(* Logix 5000 project; controller TrayLoader_EnSG vendor 1 type 14 code 156 rev 32.11; software revision 32.02; part 2 of 3 *)
(* tags used below, declared in another part *)
   blink1s : BOOL;
   Emergency : BOOL;
   Feeder_st : INT;
   FeedMotionCtrl : MOTION_INSTRUCTION;
   modRes : INT;
   mot_conv_in : INT;   // Conveyor Motor
   oddEven : BOOL;
   ons : DINT;
   ons5 : INT;
   srvMASRTray : BOOL;
   SrvMoveType : DINT;
   TrayAxis_pos : DINT;   // servo position increment
   TrayMotionCtrl : MOTION_INSTRUCTION;
   UpLift_forward : BOOL;
   UpLift_start : BOOL;
   UpLift_stop : BOOL;
   Auto : BOOL;
   auto_resumeFeeder : BOOL;
   corr_elapsedTrayPos : DINT;
   DecelDelay_t : TIMER;
   DecelVal : DINT;
   delta_TrayActualPos : DINT;
   dummy1 : BOOL;
   elapsedTrayPos : DINT;
   enableCheckingMsg : MESSAGE;
   enableHwOvertravelMsg : MESSAGE;
   EnableInputChecking : DINT;
   Fault : BOOL;
   feed_decel_spd : INT;   // mcd speed
   Feed_st : INT;
   feedDela_t : TIMER;
   FeederConvAxis : AXIS_CIP_DRIVE;
   FeedSpeed : DINT;
   finishPush_t : TIMER;
   finishPush_t0 : TIMER;
   hmi_Reset : BOOL;
   hmi_resetTrayCtr : BOOL;
   hmi_setSpeedRef : DINT;
   hmi_setSpeedRef100 : INT;
   JogPulse_m : BOOL;
   JogTime : TIMER;
   lastActualPosUnit : DINT;
   lineCtr : INT;
   man_disableUplift : BOOL;
   man_engageClutch : BOOL;
   man_feederReload : BOOL;
   man_FeedRailEnd : BOOL;
   man_JogLineDown : BOOL;
   man_JogLineUp : BOOL;
   man_ledRun : BOOL;
   man_ledStart : BOOL;
   man_ledWarning : BOOL;
   man_mot_conv_in0 : BOOL;
   man_mot_conv_in1 : BOOL;
   man_mot_conv_in2 : BOOL;
   man_mot_conv_in3 : BOOL;
   man_mot_conv_in4 : BOOL;
   man_mot_upLiftBrake : BOOL;
   man_sol_engageClutch : BOOL;
   man_SrvTrayJogMotorFwd : BOOL;
   man_srvTrayStop : BOOL;
   man_sv_exit : BOOL;
   man_sv_flipperIn : BOOL;
   man_sv_flipperOut : BOOL;
   man_sv_gripper : BOOL;
   man_sv_gripperArm : BOOL;
   man_sv_tray_in : BOOL;
   man_sv_tray_out : BOOL;
   man_UpLift_forward : BOOL;
   man_UpLift_start : BOOL;
   mot_upLiftBrake : BOOL;
   nc_ls_UpLift_bot : BOOL;
   nc_ls_UpLift_top : BOOL;
   nc_ps_exit : BOOL;   // indicate Full exit qeue
   negStepPulse : DINT;
   no_ps_FeedPlankHome : BOOL;
   no_ps_FeedRailDecel : BOOL;
   no_ps_FeedRailEndEven : BOOL;   // ps on end of FeederRail
   no_ps_FeedRailEndOdd : BOOL;
   no_ps_Serp_top : BOOL;   // ps serpentine top
   ons4 : INT;
   ons6 : DINT;
   ons7 : DINT;
   pauseFeeder : BOOL;
   ps_serp_top_t : TIMER;
   ps_serp_top_tof : TIMER;
   RailDecel : BOOL;
   Recover_UpLift : BOOL;
   ref_elpasedTrayPos : DINT;
   Reset : BOOL;
   resumeFeeder : BOOL;
   rs_sv_exit_top : BOOL;
   rs_sv_flipperOut_top : BOOL;
   rs_sv_tray_out_bot : BOOL;
   Run : BOOL;
   RunOff_t : TIMER;
   RunOn_t : TIMER;
   serp_top_t_pre : DINT;
   serp_top_tof_pre : DINT;
   ServoEndRun : BOOL;
   ServoEndRunPulse : BOOL;
   sol_engageClutch : BOOL;
   SrvTrayJogMot : BOOL;
   SrvTrayStep : BOOL;   // Servo Tray Step down
   SrvTrayStop : BOOL;
   StartSpeed : DINT;
   stepPulse : DINT;
   stepPulseAct : DINT;
   sv_exit : BOOL;
   sv_flipperIn : BOOL;
   sv_flipperOut : BOOL;
   sv_flipperOut_bot : BOOL;
   sv_flipperOut_top : BOOL;
   sv_gripper : BOOL;
   sv_gripper_bot : BOOL;   // pneu gripper
   sv_gripper_top : BOOL;
   sv_gripperArm : BOOL;
   sv_tray_in : BOOL;
   sv_tray_out : BOOL;
   sysStop : BOOL;
   total_tray : DINT;
   TrayAxis : AXIS_CIP_DRIVE;
   TraySrvBreakU : BOOL;
   TrayWComp_m : BOOL;   // Compensator mode
   Warning : BOOL;
(* MainProgram, continued *)

ROUTINE _06_BatteryFeeder   (* ladder *)
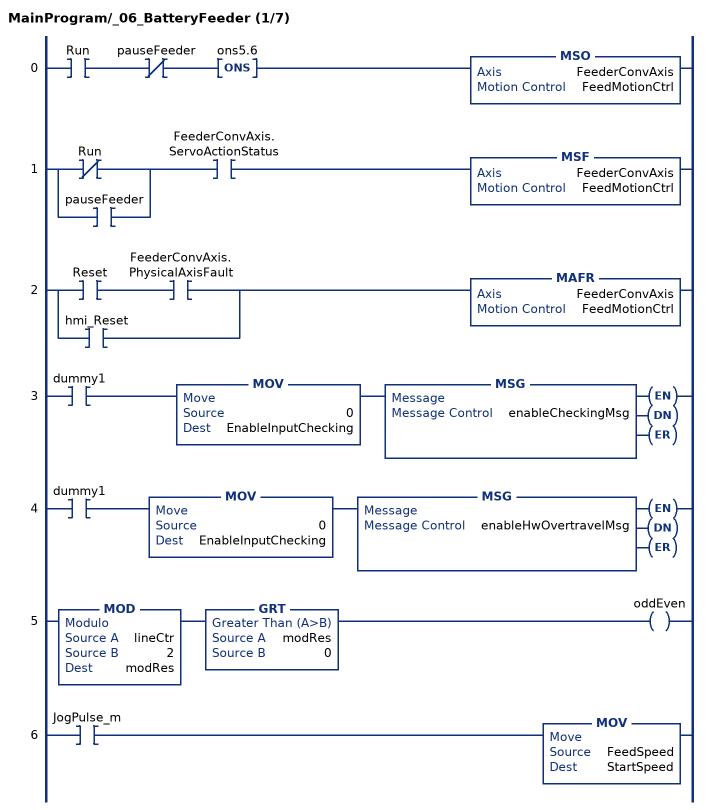
   0: XIC(Run)XIO(pauseFeeder)ONS(ons5.6)MSO(FeederConvAxis,FeedMotionCtrl);
   1: [XIO(Run) ,XIC(pauseFeeder) ]XIC(FeederConvAxis.ServoActionStatus)MSF(FeederConvAxis,FeedMotionCtrl);
   2: [XIC(Reset) XIC(FeederConvAxis.PhysicalAxisFault) ,XIC(hmi_Reset) ]MAFR(FeederConvAxis,FeedMotionCtrl);
   3: XIC(dummy1)MOV(0,EnableInputChecking)MSG(enableCheckingMsg);
   4: XIC(dummy1)MOV(0,EnableInputChecking)MSG(enableHwOvertravelMsg);
   5: MOD(lineCtr,2,modRes)GRT(modRes,0)OTE(oddEven);
   6: XIC(JogPulse_m)MOV(FeedSpeed,StartSpeed);
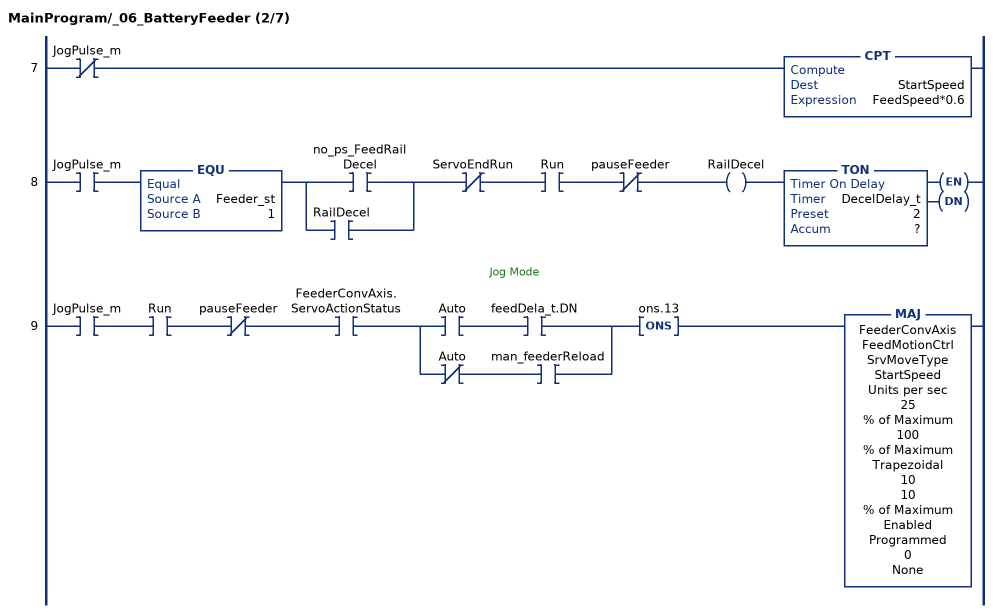
   7: XIO(JogPulse_m)CPT(StartSpeed,FeedSpeed*0.6);
   8: XIC(JogPulse_m)EQU(Feeder_st,1)[XIC(no_ps_FeedRailDecel) ,XIC(RailDecel) ]XIO(ServoEndRun)XIC(Run)XIO(pauseFeeder)OTE(RailDecel)TON(DecelDelay_t,?,?);
   // Jog Mode
   9: XIC(JogPulse_m)XIC(Run)XIO(pauseFeeder)XIC(FeederConvAxis.ServoActionStatus)[XIC(Auto) XIC(feedDela_t.DN) ,XIO(Auto) XIC(man_feederReload) ]ONS(ons.13)MAJ(FeederConvAxis,FeedMotionCtrl,SrvMoveType,StartSpeed,Units per sec,25,% of Maximum,100,% of Maximum,Trapezoidal,10,10,% of Maximum,Enabled,Programmed,0,None);
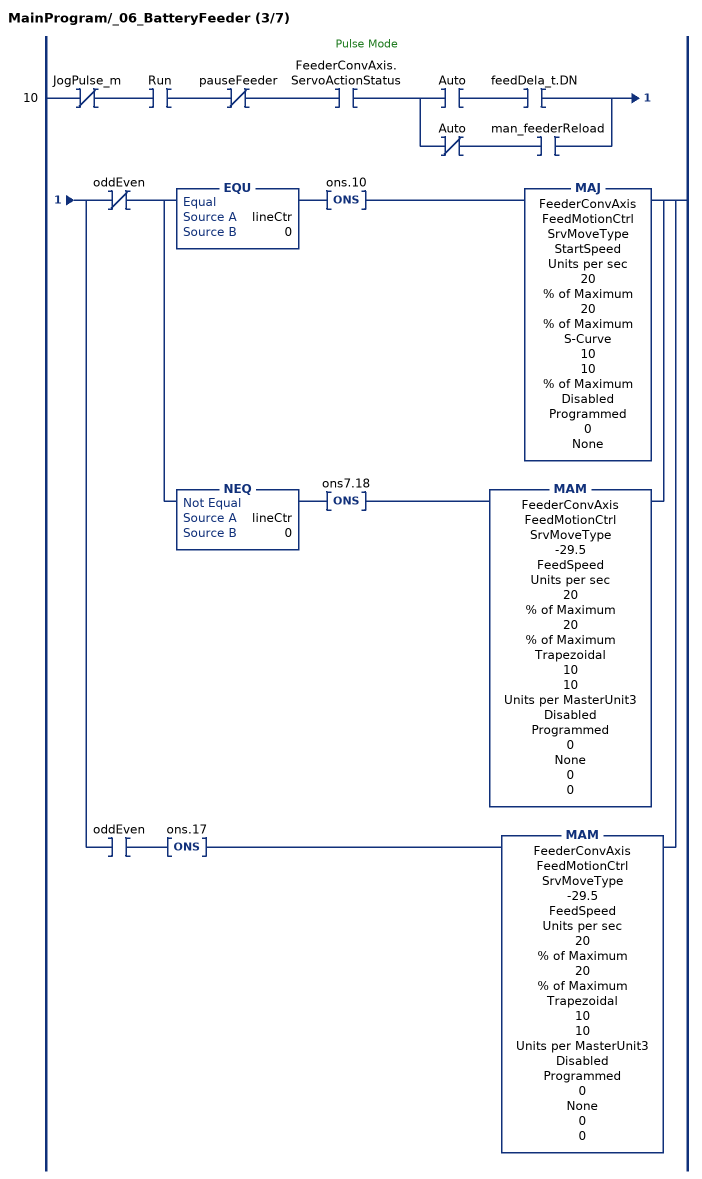
   // Pulse Mode
   10: XIO(JogPulse_m)XIC(Run)XIO(pauseFeeder)XIC(FeederConvAxis.ServoActionStatus)[XIC(Auto) XIC(feedDela_t.DN) ,XIO(Auto) XIC(man_feederReload) ][XIO(oddEven) [EQU(lineCtr,0) ONS(ons.10) MAJ(FeederConvAxis,FeedMotionCtrl,SrvMoveType,StartSpeed,Units per sec,20,% of Maximum,20,% of Maximum,S-Curve,10,10,% of Maximum,Disabled,Programmed,0,None) ,NEQ(lineCtr,0) ONS(ons7.18) MAM(FeederConvAxis,FeedMotionCtrl,SrvMoveType,-29.5,FeedSpeed,Units per sec,20,% of Maximum,20,% of Maximum,Trapezoidal,10,10,Units per MasterUnit3,Disabled,Programmed,0,None,0,0) ] ,XIC(oddEven) ONS(ons.17) MAM(FeederConvAxis,FeedMotionCtrl,SrvMoveType,-29.5,FeedSpeed,Units per sec,20,% of Maximum,20,% of Maximum,Trapezoidal,10,10,Units per MasterUnit3,Disabled,Programmed,0,None,0,0) ];
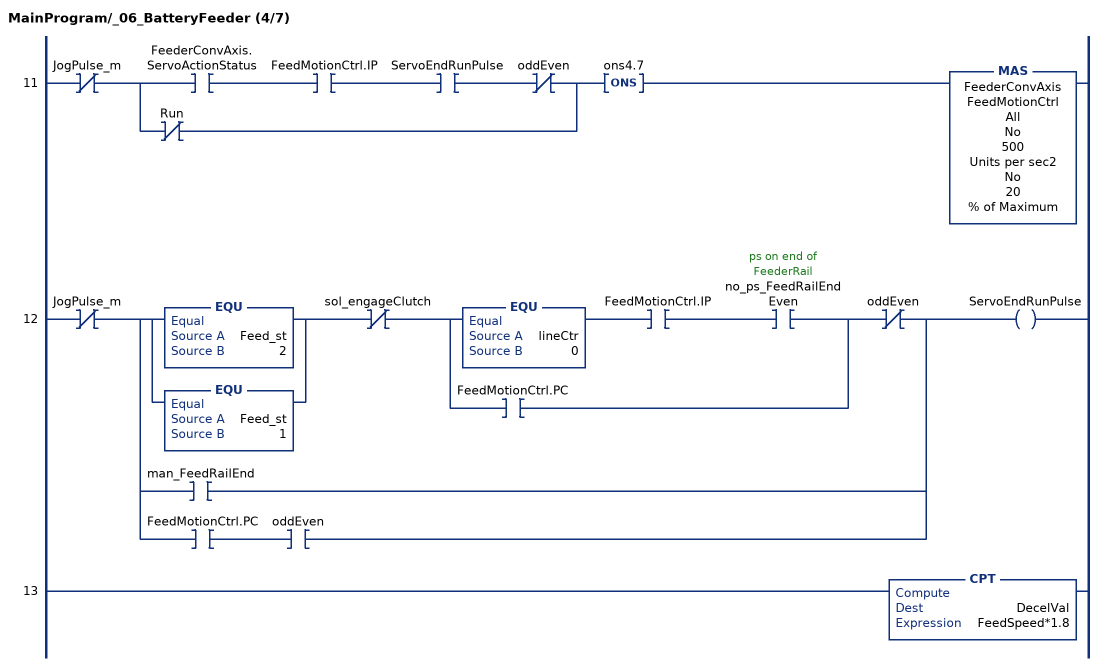
   11: XIO(JogPulse_m)[XIC(FeederConvAxis.ServoActionStatus) XIC(FeedMotionCtrl.IP) XIC(ServoEndRunPulse) XIO(oddEven) ,XIO(Run) ]ONS(ons4.7)MAS(FeederConvAxis,FeedMotionCtrl,All,No,500,Units per sec2,No,20,% of Maximum);
   12: XIO(JogPulse_m)[[EQU(Feed_st,2) ,EQU(Feed_st,1) ] XIO(sol_engageClutch) [EQU(lineCtr,0) XIC(FeedMotionCtrl.IP) XIC(no_ps_FeedRailEndEven) ,XIC(FeedMotionCtrl.PC) ] XIO(oddEven) ,XIC(man_FeedRailEnd) ,XIC(FeedMotionCtrl.PC) XIC(oddEven) ]OTE(ServoEndRunPulse);
   13: CPT(DecelVal,FeedSpeed*1.8);
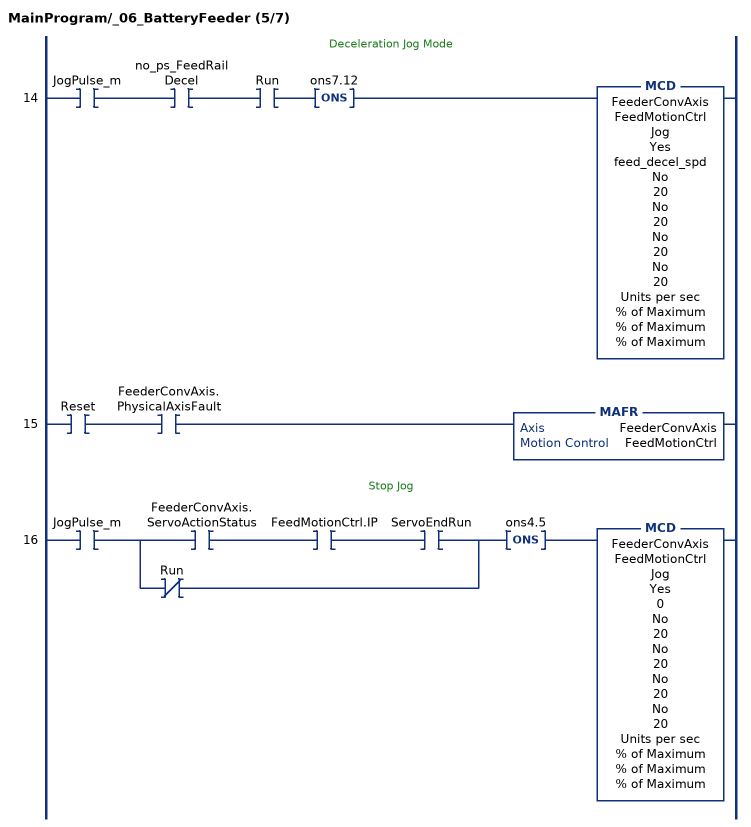
   // Deceleration Jog Mode
   14: XIC(JogPulse_m)XIC(no_ps_FeedRailDecel)XIC(Run)ONS(ons7.12)MCD(FeederConvAxis,FeedMotionCtrl,Jog,Yes,feed_decel_spd,No,20,No,20,No,20,No,20,Units per sec,% of Maximum,% of Maximum,% of Maximum);
   15: XIC(Reset)XIC(FeederConvAxis.PhysicalAxisFault)MAFR(FeederConvAxis,FeedMotionCtrl);
   // Stop Jog
   16: XIC(JogPulse_m)[XIC(FeederConvAxis.ServoActionStatus) XIC(FeedMotionCtrl.IP) XIC(ServoEndRun) ,XIO(Run) ]ONS(ons4.5)MCD(FeederConvAxis,FeedMotionCtrl,Jog,Yes,0,No,20,No,20,No,20,No,20,Units per sec,% of Maximum,% of Maximum,% of Maximum);
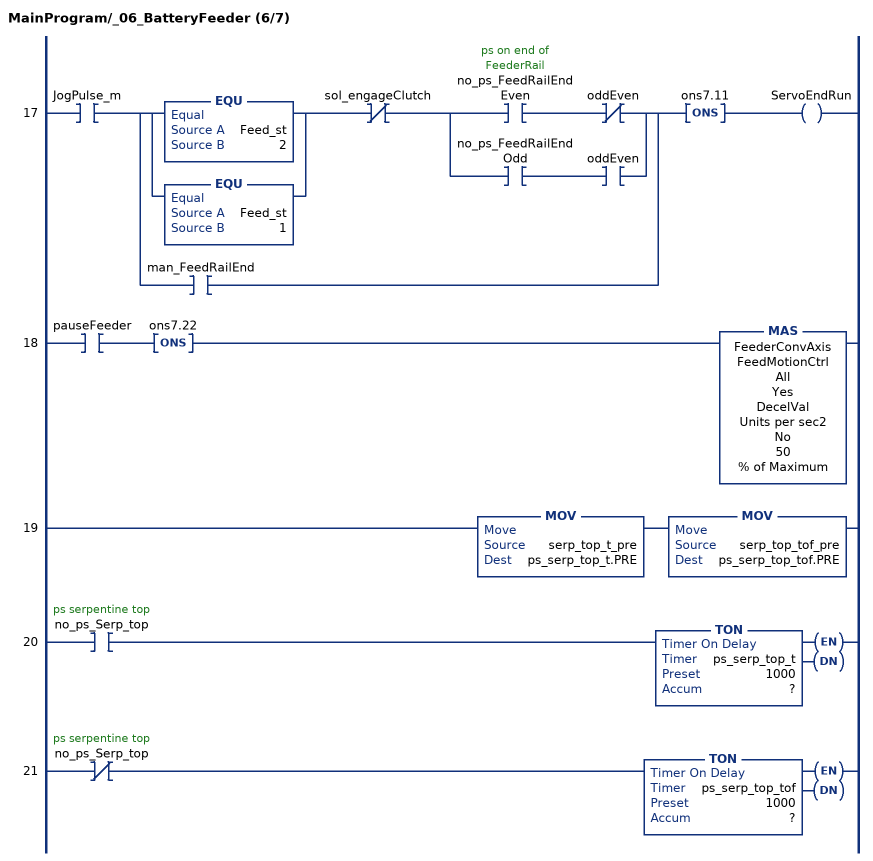
   17: XIC(JogPulse_m)[[EQU(Feed_st,2) ,EQU(Feed_st,1) ] XIO(sol_engageClutch) [XIC(no_ps_FeedRailEndEven) XIO(oddEven) ,XIC(no_ps_FeedRailEndOdd) XIC(oddEven) ] ,XIC(man_FeedRailEnd) ]ONS(ons7.11)OTE(ServoEndRun);
   18: XIC(pauseFeeder)ONS(ons7.22)MAS(FeederConvAxis,FeedMotionCtrl,All,Yes,DecelVal,Units per sec2,No,50,% of Maximum);
   19: MOV(serp_top_t_pre,ps_serp_top_t.PRE)MOV(serp_top_tof_pre,ps_serp_top_tof.PRE);
   20: XIC(no_ps_Serp_top)TON(ps_serp_top_t,?,?);
   21: XIO(no_ps_Serp_top)TON(ps_serp_top_tof,?,?);
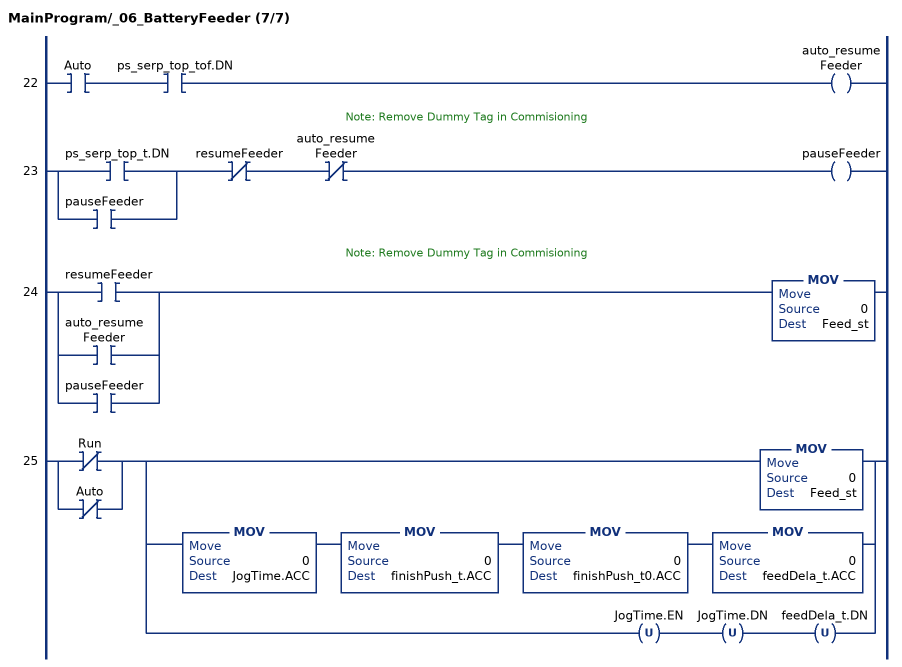
   22: XIC(Auto)XIC(ps_serp_top_tof.DN)OTE(auto_resumeFeeder);
   // Note: Remove Dummy Tag in Commisioning
   23: [XIC(ps_serp_top_t.DN) ,XIC(pauseFeeder) ]XIO(resumeFeeder)XIO(auto_resumeFeeder)OTE(pauseFeeder);
   // Note: Remove Dummy Tag in Commisioning
   24: [XIC(resumeFeeder) ,XIC(auto_resumeFeeder) ,XIC(pauseFeeder) ]MOV(0,Feed_st);
   25: [XIO(Run) ,XIO(Auto) ][MOV(0,Feed_st) ,MOV(0,JogTime.ACC) MOV(0,finishPush_t.ACC) MOV(0,finishPush_t0.ACC) MOV(0,feedDela_t.ACC) ,OTU(JogTime.EN) OTU(JogTime.DN) OTU(feedDela_t.DN) ];
END_ROUTINE

ROUTINE _07_SrvTray_lib   (* ladder *)
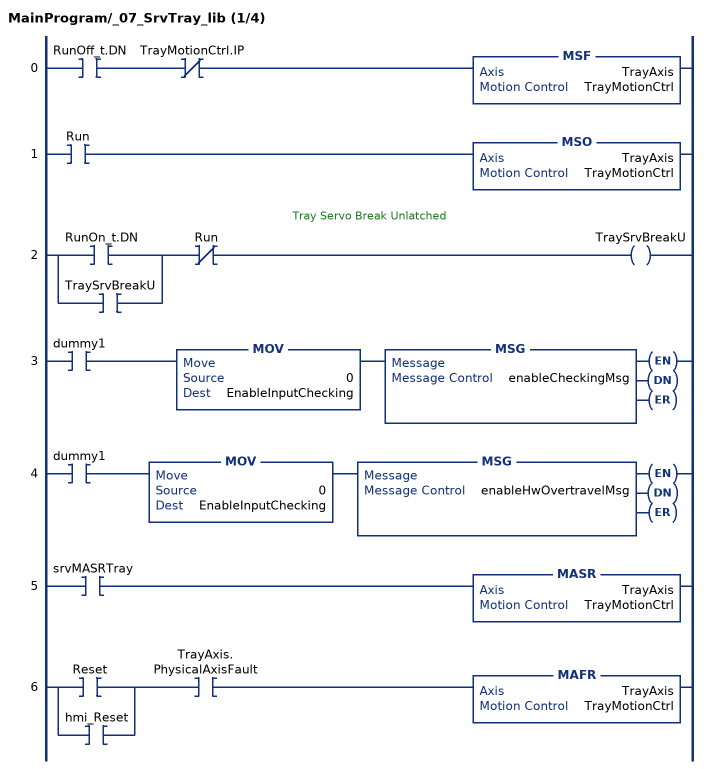
   0: XIC(RunOff_t.DN)XIO(TrayMotionCtrl.IP)MSF(TrayAxis,TrayMotionCtrl);
   1: XIC(Run)MSO(TrayAxis,TrayMotionCtrl);
   // Tray Servo Break Unlatched
   2: [XIC(RunOn_t.DN) ,XIC(TraySrvBreakU) ]XIO(Run)OTE(TraySrvBreakU);
   3: XIC(dummy1)MOV(0,EnableInputChecking)MSG(enableCheckingMsg);
   4: XIC(dummy1)MOV(0,EnableInputChecking)MSG(enableHwOvertravelMsg);
   5: XIC(srvMASRTray)MASR(TrayAxis,TrayMotionCtrl);
   6: [XIC(Reset) ,XIC(hmi_Reset) ]XIC(TrayAxis.PhysicalAxisFault)MAFR(TrayAxis,TrayMotionCtrl);
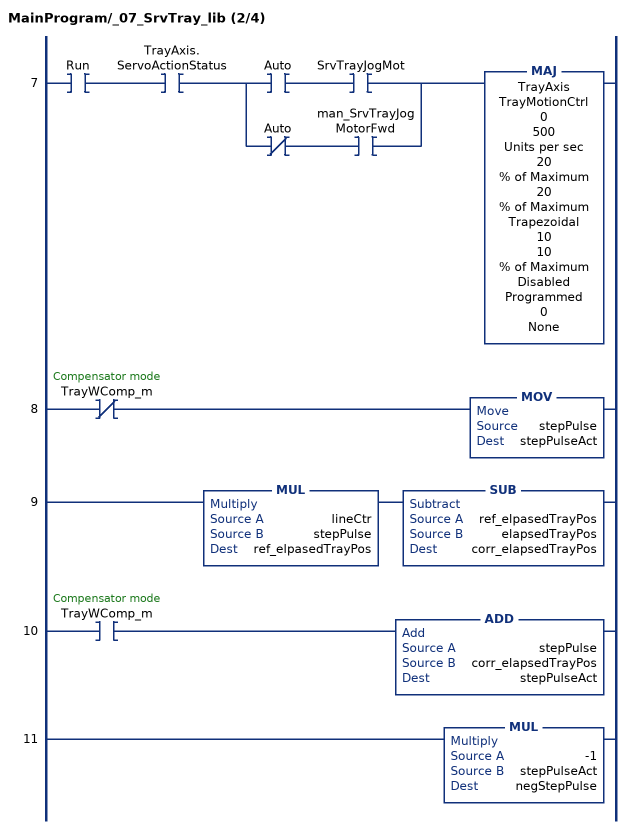
   7: XIC(Run)XIC(TrayAxis.ServoActionStatus)[XIC(Auto) XIC(SrvTrayJogMot) ,XIO(Auto) XIC(man_SrvTrayJogMotorFwd) ]MAJ(TrayAxis,TrayMotionCtrl,0,500,Units per sec,20,% of Maximum,20,% of Maximum,Trapezoidal,10,10,% of Maximum,Disabled,Programmed,0,None);
   8: XIO(TrayWComp_m)MOV(stepPulse,stepPulseAct);
   9: MUL(lineCtr,stepPulse,ref_elpasedTrayPos)SUB(ref_elpasedTrayPos,elapsedTrayPos,corr_elapsedTrayPos);
   10: XIC(TrayWComp_m)ADD(stepPulse,corr_elapsedTrayPos,stepPulseAct);
   11: MUL(-1,stepPulseAct,negStepPulse);
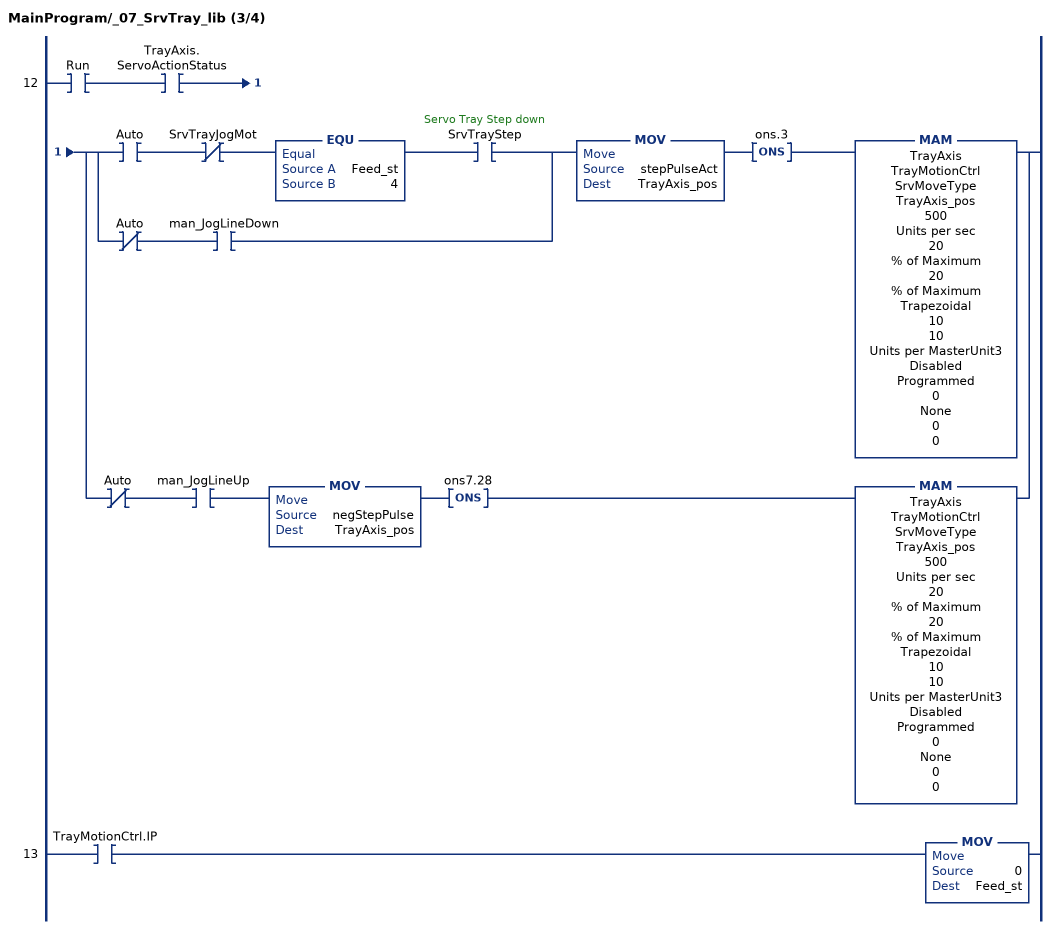
   12: XIC(Run)XIC(TrayAxis.ServoActionStatus)[[XIC(Auto) XIO(SrvTrayJogMot) EQU(Feed_st,4) XIC(SrvTrayStep) ,XIO(Auto) XIC(man_JogLineDown) ] MOV(stepPulseAct,TrayAxis_pos) ONS(ons.3) MAM(TrayAxis,TrayMotionCtrl,SrvMoveType,TrayAxis_pos,500,Units per sec,20,% of Maximum,20,% of Maximum,Trapezoidal,10,10,Units per MasterUnit3,Disabled,Programmed,0,None,0,0) ,XIO(Auto) XIC(man_JogLineUp) MOV(negStepPulse,TrayAxis_pos) ONS(ons7.28) MAM(TrayAxis,TrayMotionCtrl,SrvMoveType,TrayAxis_pos,500,Units per sec,20,% of Maximum,20,% of Maximum,Trapezoidal,10,10,Units per MasterUnit3,Disabled,Programmed,0,None,0,0) ];
   13: XIC(TrayMotionCtrl.IP)MOV(0,Feed_st);
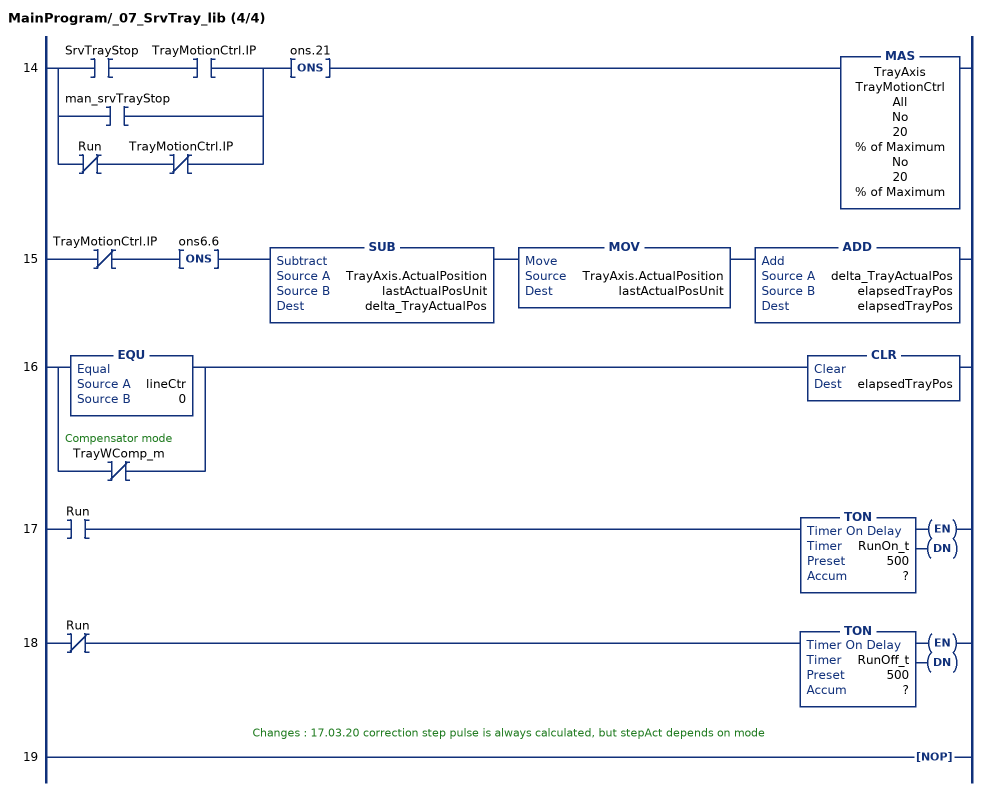
   14: [XIC(SrvTrayStop) XIC(TrayMotionCtrl.IP) ,XIC(man_srvTrayStop) ,XIO(Run) XIO(TrayMotionCtrl.IP) ]ONS(ons.21)MAS(TrayAxis,TrayMotionCtrl,All,No,20,% of Maximum,No,20,% of Maximum);
   15: XIO(TrayMotionCtrl.IP)ONS(ons6.6)SUB(TrayAxis.ActualPosition,lastActualPosUnit,delta_TrayActualPos)MOV(TrayAxis.ActualPosition,lastActualPosUnit)ADD(delta_TrayActualPos,elapsedTrayPos,elapsedTrayPos);
   16: [EQU(lineCtr,0) ,XIO(TrayWComp_m) ]CLR(elapsedTrayPos);
   17: XIC(Run)TON(RunOn_t,?,?);
   18: XIO(Run)TON(RunOff_t,?,?);
   // Changes : 17.03.20 correction step pulse is always calculated, but stepAct depends on mode
   19: NOP();
END_ROUTINE

ROUTINE _08_OutTransfer   (* ladder *)
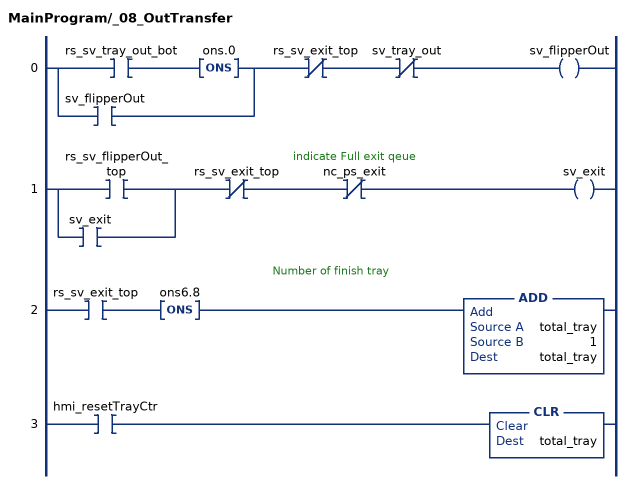
   0: [XIC(rs_sv_tray_out_bot) ONS(ons.0) ,XIC(sv_flipperOut) ]XIO(rs_sv_exit_top)XIO(sv_tray_out)OTE(sv_flipperOut);
   1: [XIC(rs_sv_flipperOut_top) ,XIC(sv_exit) ]XIO(rs_sv_exit_top)XIO(nc_ps_exit)OTE(sv_exit);
   // Number of finish tray
   2: XIC(rs_sv_exit_top)ONS(ons6.8)ADD(total_tray,1,total_tray);
   3: XIC(hmi_resetTrayCtr)CLR(total_tray);
END_ROUTINE

ROUTINE _10_Outputs   (* ladder *)
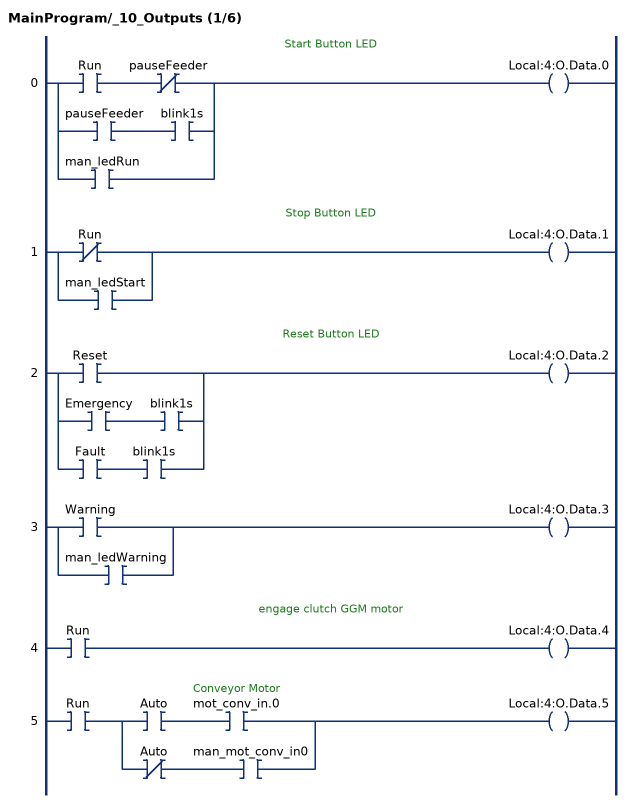
   // Start Button LED
   0: [XIC(Run) XIO(pauseFeeder) ,XIC(pauseFeeder) XIC(blink1s) ,XIC(man_ledRun) ]OTE(Local:4:O.Data.0);
   // Stop Button LED
   1: [XIO(Run) ,XIC(man_ledStart) ]OTE(Local:4:O.Data.1);
   // Reset Button LED
   2: [XIC(Reset) ,XIC(Emergency) XIC(blink1s) ,XIC(Fault) XIC(blink1s) ]OTE(Local:4:O.Data.2);
   3: [XIC(Warning) ,XIC(man_ledWarning) ]OTE(Local:4:O.Data.3);
   // engage clutch GGM motor
   4: XIC(Run)OTE(Local:4:O.Data.4);
   5: XIC(Run)[XIC(Auto) XIC(mot_conv_in.0) ,XIO(Auto) XIC(man_mot_conv_in0) ]OTE(Local:4:O.Data.5);
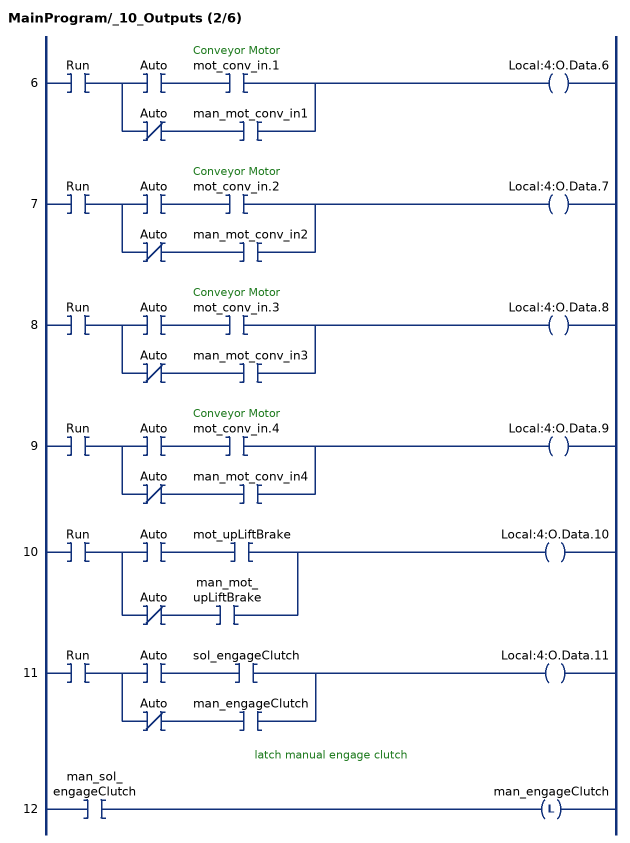
   6: XIC(Run)[XIC(Auto) XIC(mot_conv_in.1) ,XIO(Auto) XIC(man_mot_conv_in1) ]OTE(Local:4:O.Data.6);
   7: XIC(Run)[XIC(Auto) XIC(mot_conv_in.2) ,XIO(Auto) XIC(man_mot_conv_in2) ]OTE(Local:4:O.Data.7);
   8: XIC(Run)[XIC(Auto) XIC(mot_conv_in.3) ,XIO(Auto) XIC(man_mot_conv_in3) ]OTE(Local:4:O.Data.8);
   9: XIC(Run)[XIC(Auto) XIC(mot_conv_in.4) ,XIO(Auto) XIC(man_mot_conv_in4) ]OTE(Local:4:O.Data.9);
   10: XIC(Run)[XIC(Auto) XIC(mot_upLiftBrake) ,XIO(Auto) XIC(man_mot_upLiftBrake) ]OTE(Local:4:O.Data.10);
   11: XIC(Run)[XIC(Auto) XIC(sol_engageClutch) ,XIO(Auto) XIC(man_engageClutch) ]OTE(Local:4:O.Data.11);
   // latch manual engage clutch
   12: XIC(man_sol_engageClutch)OTL(man_engageClutch);
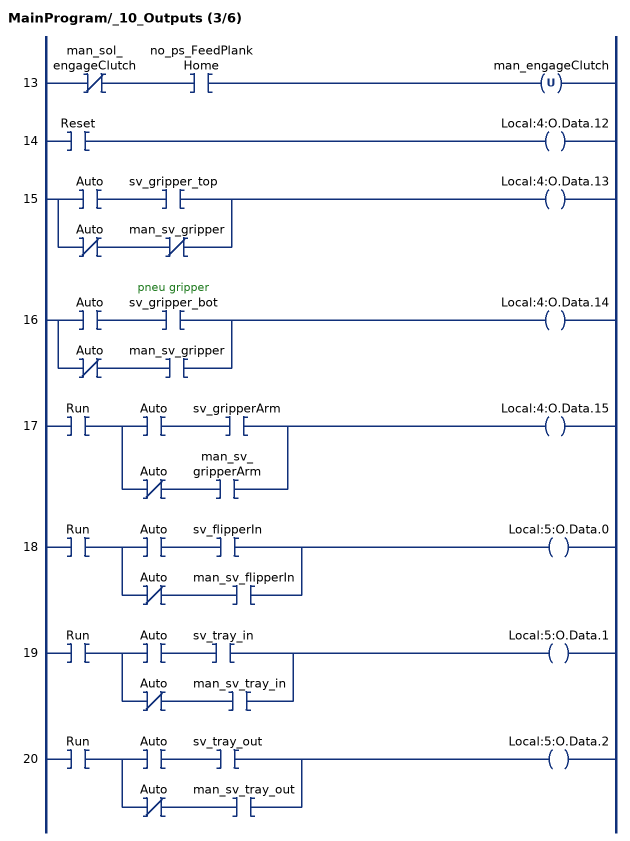
   13: XIO(man_sol_engageClutch)XIC(no_ps_FeedPlankHome)OTU(man_engageClutch);
   14: XIC(Reset)OTE(Local:4:O.Data.12);
   15: [XIC(Auto) XIC(sv_gripper_top) ,XIO(Auto) XIO(man_sv_gripper) ]OTE(Local:4:O.Data.13);
   16: [XIC(Auto) XIC(sv_gripper_bot) ,XIO(Auto) XIC(man_sv_gripper) ]OTE(Local:4:O.Data.14);
   17: XIC(Run)[XIC(Auto) XIC(sv_gripperArm) ,XIO(Auto) XIC(man_sv_gripperArm) ]OTE(Local:4:O.Data.15);
   18: XIC(Run)[XIC(Auto) XIC(sv_flipperIn) ,XIO(Auto) XIC(man_sv_flipperIn) ]OTE(Local:5:O.Data.0);
   19: XIC(Run)[XIC(Auto) XIC(sv_tray_in) ,XIO(Auto) XIC(man_sv_tray_in) ]OTE(Local:5:O.Data.1);
   20: XIC(Run)[XIC(Auto) XIC(sv_tray_out) ,XIO(Auto) XIC(man_sv_tray_out) ]OTE(Local:5:O.Data.2);
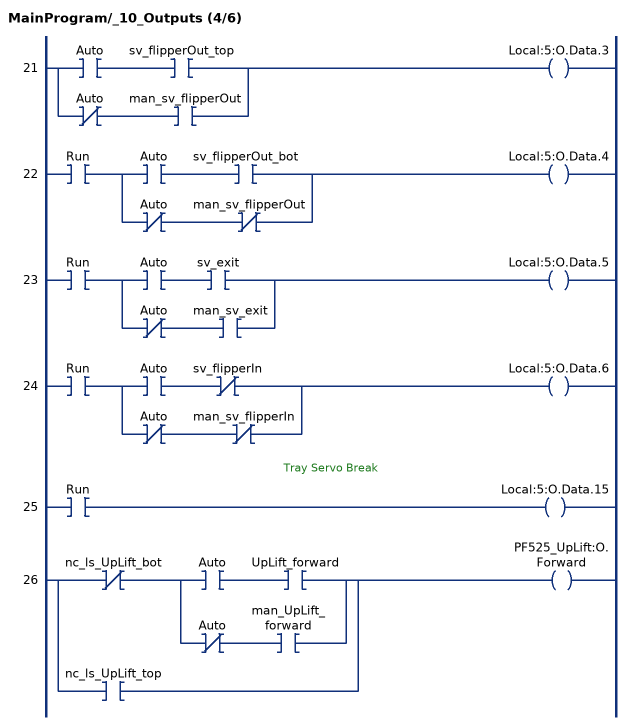
   21: [XIC(Auto) XIC(sv_flipperOut_top) ,XIO(Auto) XIC(man_sv_flipperOut) ]OTE(Local:5:O.Data.3);
   22: XIC(Run)[XIC(Auto) XIC(sv_flipperOut_bot) ,XIO(Auto) XIO(man_sv_flipperOut) ]OTE(Local:5:O.Data.4);
   23: XIC(Run)[XIC(Auto) XIC(sv_exit) ,XIO(Auto) XIC(man_sv_exit) ]OTE(Local:5:O.Data.5);
   24: XIC(Run)[XIC(Auto) XIO(sv_flipperIn) ,XIO(Auto) XIO(man_sv_flipperIn) ]OTE(Local:5:O.Data.6);
   // Tray Servo Break
   25: XIC(Run)OTE(Local:5:O.Data.15);
   26: [XIO(nc_ls_UpLift_bot) [XIC(Auto) XIC(UpLift_forward) ,XIO(Auto) XIC(man_UpLift_forward) ] ,XIC(nc_ls_UpLift_top) ]OTE(PF525_UpLift:O.Forward);
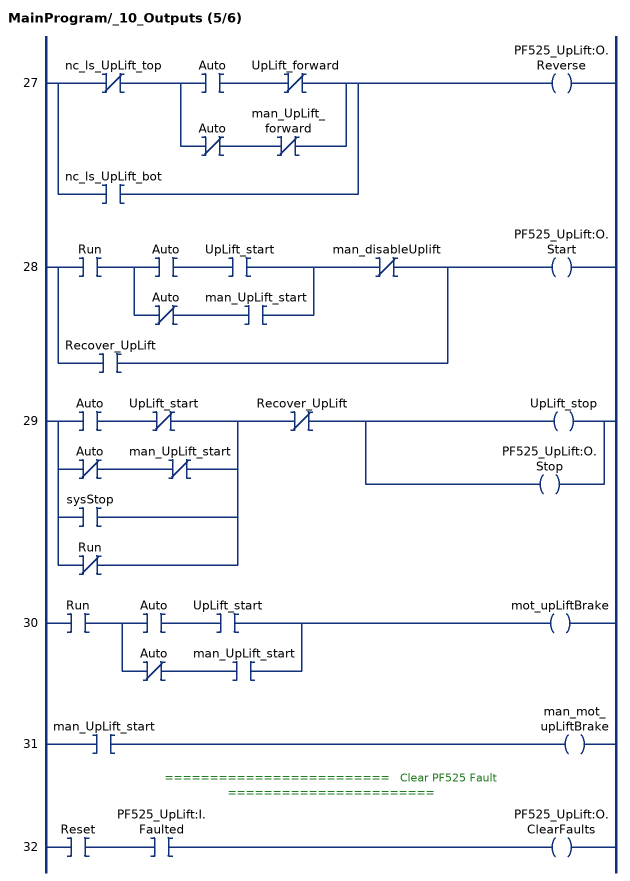
   27: [XIO(nc_ls_UpLift_top) [XIC(Auto) XIO(UpLift_forward) ,XIO(Auto) XIO(man_UpLift_forward) ] ,XIC(nc_ls_UpLift_bot) ]OTE(PF525_UpLift:O.Reverse);
   28: [XIC(Run) [XIC(Auto) XIC(UpLift_start) ,XIO(Auto) XIC(man_UpLift_start) ] XIO(man_disableUplift) ,XIC(Recover_UpLift) ]OTE(PF525_UpLift:O.Start);
   29: [XIC(Auto) XIO(UpLift_start) ,XIO(Auto) XIO(man_UpLift_start) ,XIC(sysStop) ,XIO(Run) ]XIO(Recover_UpLift)[OTE(UpLift_stop) ,OTE(PF525_UpLift:O.Stop) ];
   30: XIC(Run)[XIC(Auto) XIC(UpLift_start) ,XIO(Auto) XIC(man_UpLift_start) ]OTE(mot_upLiftBrake);
   31: XIC(man_UpLift_start)OTE(man_mot_upLiftBrake);
   // =========================   Clear PF525 Fault   =======================
   32: XIC(Reset)XIC(PF525_UpLift:I.Faulted)OTE(PF525_UpLift:O.ClearFaults);
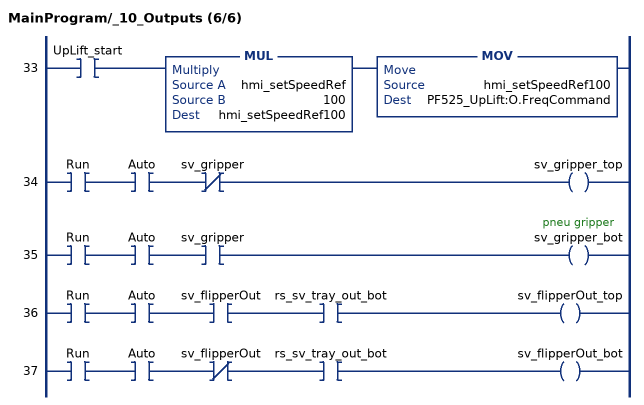
   33: XIC(UpLift_start)MUL(hmi_setSpeedRef,100,hmi_setSpeedRef100)MOV(hmi_setSpeedRef100,PF525_UpLift:O.FreqCommand);
   34: XIC(Run)XIC(Auto)XIO(sv_gripper)OTE(sv_gripper_top);
   35: XIC(Run)XIC(Auto)XIC(sv_gripper)OTE(sv_gripper_bot);
   36: XIC(Run)XIC(Auto)XIC(sv_flipperOut)XIC(rs_sv_tray_out_bot)OTE(sv_flipperOut_top);
   37: XIC(Run)XIC(Auto)XIO(sv_flipperOut)XIC(rs_sv_tray_out_bot)OTE(sv_flipperOut_bot);
END_ROUTINE
